PROGRAM prgPersistent
VAR
	fbUSV		: FB_WritePersistentData_CX81xx;
	
	fb_Reboot		: NT_reboot;
	m_Reboot		: BOOL:=FALSE;
	Int_LiveCount_1min	:INT; 							//{#lynus.ag#()}
	ton_LiveCount	:TON;	
	int_liveCount		:INT;				//{#lynus.ag#()}
END_VAR

fbUSV(
	eSaveModeData:= eUSVSaveMode.eSaveWhenPowerfail, 
	bLoadPersistentDataOk=> , 
	bPowerFailDetect=> , 
	bError=> , 
	bySaveProcess=> , 
	dwStorageLast24h=> , 
	udiErrorCode=> );
	
	
fb_Reboot(	netid := '',
			delay := 2,
			start := m_Reboot);

// 1 min live count
ton_LiveCount(PT:=T#1M);
IF ton_LiveCount.Q THEN
	Int_LiveCount_1min := Int_LiveCount_1min + 1;
	ton_LiveCount.IN := FALSE;
ELSE
	ton_LiveCount.IN := TRUE;
END_IF
// livecount
int_liveCount := int_liveCount+1;

END_PROGRAM

(* stored: Version 1.1.0.1, ProductVersion 3.1.4024.12
   POU prgPersistent: Id {ccd67b8a-d866-4216-a145-3575a5a9eafe}, SpecialFunc None *)
